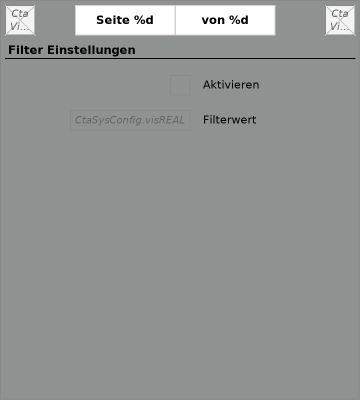
VISUALIZATION VIS_SENSOR_PARAMETER_FILTER  // 360x400
VAR_INPUT
  	ITF_SENSORIN	:	ITF_SENSOR;
END_VAR
VAR
    uiPage  :   UINT;
    uiMin   :   UINT    := 0;
    uiMax   :   UINT    := 0;
END_VAR
    Image (5,5 30x30), invisible if: uiPage = uiMin, image: CtaVisSymbols.ImagePool.arrow-left_square
        OnMouseClick: execute {
            uiPage := uiPage - 1;
            IF uiPage <= uiMin THEN
                uiPage := uiMin;
            END_IF;
        }
    Image (325,5 30x30), invisible if: uiPage = uiMax, image: CtaVisSymbols.ImagePool.arrow-right_square
        OnMouseClick: execute {
            uiPage := uiPage + 1;
            IF uiPage >= uiMax THEN
                uiPage := uiMax;
            END_IF;
        }
    Frame (0,40 360x360), frame switch variable: uiPage
        shows VIS_SENSOR_PARAMETER_FILTER_1(ITF_SENSORIN := ITF_SENSORIN)
        shows AT_ParameterIO1(ITF_Parameter := ITF_Parameter)
    Textfield (175,5 100x30), "von %d", text variable: uiMax
    Textfield (75,5 100x30), "Seite %d", text variable: uiPage
END_VISUALIZATION

// 40 Visualizations/POPUP/PARAMETER/SENSOR_Filter/VIS_SENSOR_PARAMETER_FILTER_1
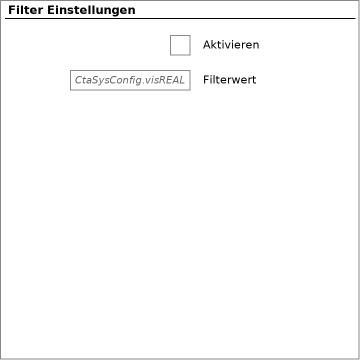
VISUALIZATION VIS_SENSOR_PARAMETER_FILTER_1  // 360x360
VAR_INPUT
   	ITF_SENSORIN	:	ITF_SENSOR;
END_VAR
    Label (5,0 350x20), "Filter Einstellungen"
    Line (5,18) (355,18)
    Frame (170,35 20x20)
        shows CtaSysConfig.visBOOL(visfbBOOLIn := ITF_SENSORIN.P_scFilter_fbxEnabled)
    Label (200,35 150x20), "Aktivieren"
    Frame (70,70 120x20)
        shows CtaSysConfig.visREAL(visfbREALIn := ITF_SENSORIN.P_scFilter_fbrValue)
    Label (200,70 150x20), "Filterwert"
END_VISUALIZATION

// 40 Visualizations/POPUP/PARAMETER/SENSOR_InfluxDb/VIS_SENSOR_PARAMETER_TRENDLOG
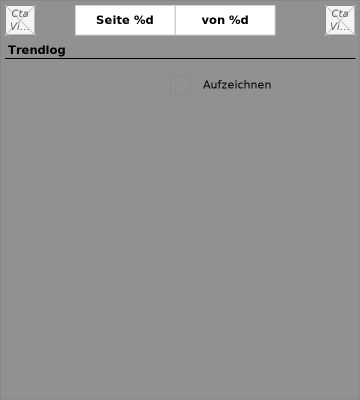
VISUALIZATION VIS_SENSOR_PARAMETER_TRENDLOG  // 360x400
VAR_INPUT
   	ITF_SENSORIN	:	ITF_SENSOR;
END_VAR
VAR
    uiPage  :   UINT;
    uiMin   :   UINT    := 0;
    uiMax   :   UINT    := 0;
END_VAR
    Image (5,5 30x30), invisible if: uiPage = uiMin, image: CtaVisSymbols.ImagePool.arrow-left_square
        OnMouseClick: execute {
            uiPage := uiPage - 1;
            IF uiPage <= uiMin THEN
                uiPage := uiMin;
            END_IF;
        }
    Image (325,5 30x30), invisible if: uiPage = uiMax, image: CtaVisSymbols.ImagePool.arrow-right_square
        OnMouseClick: execute {
            uiPage := uiPage + 1;
            IF uiPage >= uiMax THEN
                uiPage := uiMax;
            END_IF;
        }
    Frame (0,40 360x360), frame switch variable: uiPage
        shows VIS_SENSOR_PARAMETER_TRENDLOG0(ITF_SENSORIN := ITF_SENSORIN)
        shows AT_ParameterIO1(ITF_Parameter := ITF_Parameter)
        pReferences[0]: ITF_Parameter=ITF_Parameter
    Textfield (75,5 100x30), "Seite %d", text variable: uiPage
    Textfield (175,5 100x30), "von %d", text variable: uiMax
END_VISUALIZATION

// 40 Visualizations/POPUP/PARAMETER/SENSOR_InfluxDb/VIS_SENSOR_PARAMETER_TRENDLOG0
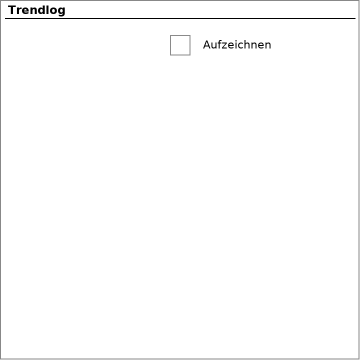
VISUALIZATION VIS_SENSOR_PARAMETER_TRENDLOG0  // 360x360
VAR_INPUT
    ITF_SENSORIN	:	ITF_SENSOR;
END_VAR
    Frame (170,35 20x20)
        shows CtaSysConfig.visBOOL(visfbBOOLIn := ITF_SENSORIN.P_scInfluxDb_fbxEnable)
    Label (200,35 150x20), "Aufzeichnen"
    Label (5,0 350x20), "Trendlog"
    Line (5,18) (355,18)
END_VISUALIZATION

// 40 Visualizations/POPUP/PARAMETER/SENSOR_ReportManagement/Sensor_LowWarning_Param
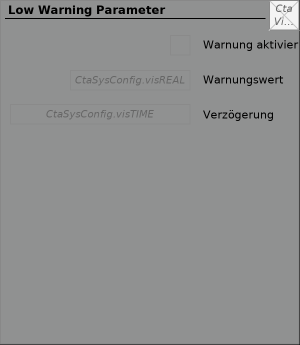
VISUALIZATION Sensor_LowWarning_Param  // 300x345
VAR_INPUT
	ITF_SENSORIN	:	ITF_SENSOR;
END_VAR
VAR_IN_OUT
    xShow   :   BOOL;
END_VAR
    Rectangle (0,0 300x345)
    Image (269,0 30x30), image: CtaVisSymbols.ImagePool.close_solo_black
        OnMouseClick: execute { xShow := FALSE; }
    Label (5,0 198x20), "Low Warning Parameter"
    Line (5,18) (265,18)
    Label (200,35 100x20), "Warnung aktiviert"
    Frame (170,35 20x20)
        shows CtaSysConfig.visBOOL(visfbBOOLIn := ITF_SENSORIN.P_scLoWarning_fbxDoesWarning)
    Label (200,70 100x20), "Warnungswert"
    Frame (70,70 120x20), invisible if: (ITF_SENSORIN.proValueInputType = enInputType.DigitalInput) OR (ITF_SENSORIN.proValueInputType = enInputType.Digital_ITF_Input)
        shows CtaSysConfig.visREAL(visfbREALIn := ITF_SENSORIN.P_scLoWarning_fbrValue)
    Label (200,105 100x20), "Verzögerung"
    Frame (10,104 180x20)
        shows CtaSysConfig.visTIME(visfbTIMEIn := ITF_SENSORIN.P_scLoWarning_fbtDelayTillWarning)
END_VISUALIZATION

// 40 Visualizations/ICON/SENSOR_FLAT/SENSOR_FLAT_TXT_RIGHT/ABOVE/VIS_SENSOR_FLAT_RigthAboveCheckQuerry
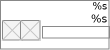
VISUALIZATION VIS_SENSOR_FLAT_RigthAboveCheckQuerry  // 110x50
VAR_INPUT
    ITF_SENSOR_IN   :   ITF_SENSOR;
	stExklParameter	:	STRING [40];
END_VAR
    Frame (0,0 110x50)
        shows VIS_SENSOR_FLAT_RigthAboveCheckIsEnabled(ITF_SENSOR_IN := ITF_SENSOR_IN, stExklParameter := stExklParameter)
END_VISUALIZATION

// 40 Visualizations/ICON/SENSOR_ROUND/SENSOR_ROUNF_TXT_LEFT/ABOVE/VIS_SENSOR_ROUND_LEFT_ABOVE
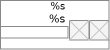
VISUALIZATION VIS_SENSOR_ROUND_LEFT_ABOVE  // 110x50
VAR_INPUT
    ITF_SENSOR_IN   :   ITF_SENSOR;	
END_VAR
VAR_INPUT CONSTANT	
	stExklParameter	:	STRING [40] := ' ';	
END_VAR
VAR CONSTANT
	uiIconnr		:	UINT := 6;
END_VAR
    Frame (0,0 110x50), invisible if: NOT fcCheckQuerryAndIconReturn(_ITF_IN := ITF_SENSOR_IN, _uiIconNr_IN := uiIconNr)
        shows VIS_SENSOR_ROUND_LeftAboveCheckQuerry(ITF_SENSOR_IN := ITF_SENSOR_IN, stExklParameter := stExklParameter)
END_VISUALIZATION

// 40 Visualizations/ICON/SENSOR_ROUND/SENSOR_ROUNF_TXT_LEFT/ABOVE/VIS_SENSOR_ROUND_LeftAboveCheckIsEnabled
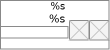
VISUALIZATION VIS_SENSOR_ROUND_LeftAboveCheckIsEnabled  // 110x50
VAR_INPUT
    ITF_SENSOR_IN   :   ITF_SENSOR;
	stExklParameter	:	STRING [40];	
END_VAR
    Frame (69,20 40x20), invisible if: NOT ITF_SENSOR_IN.proIsEnabled
        shows SensorRound(ITF_SENSORIN := ITF_SENSOR_IN)
    Frame (0,0 68x40), invisible if: NOT ITF_SENSOR_IN.proIsEnabled
        shows ValueUpDwn(ITF_SENSORIN := ITF_SENSOR_IN, uiTextAusrichtung := 6)
    Rectangle (0,0 110x50)
        OnMouseClick:  Dialog=POPUP_SENSOR, Parameters={stExklParameter: stExklParameter, ITF_SENSORIN: ITF_SENSOR_IN, uiPopUpGruppe: 0}, OpenCentered=True
END_VISUALIZATION

// 40 Visualizations/ICON/SENSOR_ROUND/SENSOR_ROUNF_TXT_LEFT/ABOVE/VIS_SENSOR_ROUND_LeftAboveCheckQuerry
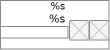
VISUALIZATION VIS_SENSOR_ROUND_LeftAboveCheckQuerry  // 110x50
VAR_INPUT
    ITF_SENSOR_IN   :   ITF_SENSOR;
	stExklParameter	:	STRING [40];	
END_VAR
    Frame (0,0 110x50)
        shows VIS_SENSOR_ROUND_LeftAboveCheckIsEnabled(ITF_SENSOR_IN := ITF_SENSOR_IN, stExklParameter := stExklParameter)
END_VISUALIZATION

// 40 Visualizations/ICON/SENSOR_ROUND/SENSOR_ROUND_TXT_RIGHT/ABOVE/VIS_SENSOR_ROUND_RIGHT_ABOVE
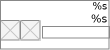
VISUALIZATION VIS_SENSOR_ROUND_RIGHT_ABOVE  // 110x50
VAR_INPUT
    ITF_SENSOR_IN   :   ITF_SENSOR;	
END_VAR
VAR_INPUT CONSTANT	
	stExklParameter	:	STRING [40] := ' ';	
END_VAR
VAR CONSTANT
	uiIconNr		:	UINT := 4;
END_VAR
    Frame (0,0 110x50), invisible if: NOT fcCheckQuerryAndIconReturn(_ITF_IN := ITF_SENSOR_IN, _uiIconNr_IN := uiIconNr)
        shows VIS_SENSOR_ROUND_RightAboveCheckQuerry(ITF_SENSOR_IN := ITF_SENSOR_IN, stExklParameter := stExklParameter)
END_VISUALIZATION

// 40 Visualizations/ICON/SENSOR_ROUND/SENSOR_ROUND_TXT_RIGHT/ABOVE/VIS_SENSOR_ROUND_RightAboveCheckIsEnabled
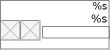
VISUALIZATION VIS_SENSOR_ROUND_RightAboveCheckIsEnabled  // 110x50
VAR_INPUT
    ITF_SENSOR_IN   :   ITF_SENSOR;
	stExklParameter	:	STRING [40];	
END_VAR
    Frame (0,20 40x20), invisible if: NOT ITF_SENSOR_IN.proIsEnabled
        shows SensorRound(ITF_SENSORIN := ITF_SENSOR_IN)
    Frame (42,0 68x40), invisible if: NOT ITF_SENSOR_IN.proIsEnabled
        shows ValueUpDwn(ITF_SENSORIN := ITF_SENSOR_IN, uiTextAusrichtung := 4)
    Rectangle (0,0 110x50)
        OnMouseClick:  Dialog=POPUP_SENSOR, Parameters={stExklParameter: stExklParameter, ITF_SENSORIN: ITF_SENSOR_IN, uiPopUpGruppe: 0}, OpenCentered=True
END_VISUALIZATION

// 40 Visualizations/ICON/SENSOR_ROUND/SENSOR_ROUND_TXT_RIGHT/ABOVE/VIS_SENSOR_ROUND_RightAboveCheckQuerry
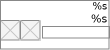
VISUALIZATION VIS_SENSOR_ROUND_RightAboveCheckQuerry  // 110x50
VAR_INPUT
    ITF_SENSOR_IN   :   ITF_SENSOR;
	stExklParameter	:	STRING [40];	
END_VAR
    Frame (0,0 110x50)
        shows VIS_SENSOR_ROUND_RightAboveCheckIsEnabled(ITF_SENSOR_IN := ITF_SENSOR_IN, stExklParameter := stExklParameter)
END_VISUALIZATION

// 40 Visualizations/ICON/SENSOR_FLAT/SENSOR_FLAT_TXT_RIGHT/BELOW/VIS_SENSOR_FLAT_RIGHT_BELOW
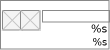
VISUALIZATION VIS_SENSOR_FLAT_RIGHT_BELOW  // 110x50
VAR_INPUT
    ITF_SENSOR_IN   :   ITF_SENSOR;	
END_VAR
VAR_INPUT CONSTANT	
	stExklParameter	:	STRING [40] := ' ';	
END_VAR
VAR CONSTANT
	uiIconNr		:	UINT := 3;
END_VAR
    Frame (0,0 110x50), invisible if: NOT fcCheckQuerryAndIconReturn(_ITF_IN := ITF_SENSOR_IN, _uiIconNr_IN := uiIconNr)
        shows VIS_SENSOR_FLAT_RigthBelowCheckQuerry(ITF_SENSOR_IN := ITF_SENSOR_IN, stExklParameter := stExklParameter)
END_VISUALIZATION

// 40 Visualizations/ICON/SENSOR_FLAT/SENSOR_FLAT_TXT_RIGHT/BELOW/VIS_SENSOR_FLAT_RigthBelowCheckIsEnabled
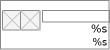
VISUALIZATION VIS_SENSOR_FLAT_RigthBelowCheckIsEnabled  // 110x50
VAR_INPUT
    ITF_SENSOR_IN   :   ITF_SENSOR;
	stExklParameter	:	STRING [40];	
END_VAR
    Frame (2,10 38x20), invisible if: NOT ITF_SENSOR_IN.proIsEnabled
        shows SensorFlat(ITF_SENSORIN := ITF_SENSOR_IN)
    Frame (42,10 68x40), invisible if: NOT ITF_SENSOR_IN.proIsEnabled
        shows ValueDwnUp(ITF_SENSORIN := ITF_SENSOR_IN, uiTextAusrichtung := 4)
    Rectangle (0,0 110x50)
        OnMouseClick:  Dialog=POPUP_SENSOR, Parameters={stExklParameter: stExklParameter, ITF_SENSORIN: ITF_SENSOR_IN, uiPopUpGruppe: 0}, OpenCentered=True
END_VISUALIZATION

// 40 Visualizations/ICON/SENSOR_FLAT/SENSOR_FLAT_TXT_RIGHT/BELOW/VIS_SENSOR_FLAT_RigthBelowCheckQuerry
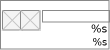
VISUALIZATION VIS_SENSOR_FLAT_RigthBelowCheckQuerry  // 110x50
VAR_INPUT
    ITF_SENSOR_IN   :   ITF_SENSOR;	
	stExklParameter	:	STRING [40];	
END_VAR
    Frame (0,0 110x50)
        shows VIS_SENSOR_FLAT_RigthBelowCheckIsEnabled(ITF_SENSOR_IN := ITF_SENSOR_IN, stExklParameter := stExklParameter)
END_VISUALIZATION

// 40 Visualizations/ICON/SENSOR_ROUND/SENSOR_ROUND_TXT_RIGHT/BELOW/VIS_SENSOR_ROUND_RIGHT_BELOW
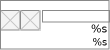
VISUALIZATION VIS_SENSOR_ROUND_RIGHT_BELOW  // 110x50
VAR_INPUT
    ITF_SENSOR_IN   :   ITF_SENSOR;	
END_VAR
VAR_INPUT CONSTANT	
	stExklParameter	:	STRING [40] := ' ';	
END_VAR
VAR CONSTANT
	uiIconNr		:	UINT := 5;
END_VAR
    Frame (0,0 110x50), invisible if: NOT fcCheckQuerryAndIconReturn(_ITF_IN := ITF_SENSOR_IN, _uiIconNr_IN := uiIconNr)
        shows VIS_SENSOR_ROUND_RightBelowCheckQuerry(ITF_SENSOR_IN := ITF_SENSOR_IN, stExklParameter := stExklParameter)
END_VISUALIZATION

// 40 Visualizations/ICON/SENSOR_BASE/ICON/Value/ValueDwnUp
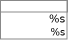
VISUALIZATION ValueDwnUp  // 68x40
VAR_INPUT
    ITF_SENSORIN   :   ITF_SENSOR;	
END_VAR
VAR_INPUT CONSTANT
    uiTextAusrichtung   : UINT := 4;    // 0 = Oben links | 1 = Horizontal zentriert | 2 = Rechts | 4 = Vertikal zentriert | 8 = Unten
END_VAR
    Frame (0,0 68x12)
        shows CtaSysSensorReCalculation.ValueRC(ITF_SENSOR_RE_CALCULATE := ITF_SENSORIN.ITF_RC, uiTextAusrichtung := uiTextAusrichtung)
    Textfield (0,13 68x12), "%s", text variable: ITF_SENSORIN.proSoftwareValue
        p3718999670: uiTextAusrichtung
    Textfield (0,26 68x12), "%s", text variable: ITF_SENSORIN.proGetBMK, invisible if: ITF_SENSORIN.proNoBmkInList
        p3718999670: uiTextAusrichtung
END_VISUALIZATION

// 40 Visualizations/ICON/SENSOR_BASE/ICON/Round/SensorRound
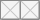
VISUALIZATION SensorRound  // 40x20
VAR_INPUT
    ITF_SENSORIN   :   ITF_SENSOR;	
END_VAR
    Ellipse (10,0 20x20), colour toggle: ITF_SENSORIN.proAcknowlege, invisible if: ITF_SENSORIN.proIsError
    Ellipse (10,0 20x20), colour toggle: ITF_SENSORIN.proIsError
    Image (0,0 20x20), invisible if: NOT ITF_SENSORIN.proIsWarning, image: CtaVisSymbols.ImagePool.CtaWarning
    Image (20,0 20x20), invisible if: NOT ITF_SENSORIN.proIsHandOnOrOff, image: CtaVisSymbols.ImagePool.front_hand_Yellow
    Image (20,0 20x20), invisible if: NOT ITF_SENSORIN.proHandOff, image: CtaVisSymbols.ImagePool.front_hand_Yellow_Off
END_VISUALIZATION

// 40 Visualizations/ICON/SENSOR_ROUND/SENSOR_ROUND_TXT_RIGHT/BELOW/VIS_SENSOR_ROUND_RightBelowCheckQuerry
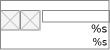
VISUALIZATION VIS_SENSOR_ROUND_RightBelowCheckQuerry  // 110x50
VAR_INPUT
    ITF_SENSOR_IN   :   ITF_SENSOR;
	stExklParameter	:	STRING [40];	
END_VAR
    Frame (0,0 110x50)
        shows VIS_SENSOR_ROUND_RightBelowCheckIsEnabled(ITF_SENSOR_IN := ITF_SENSOR_IN, stExklParameter := stExklParameter)
END_VISUALIZATION

// 40 Visualizations/ICON/SENSOR_ROUND/SENSOR_ROUND_TXT_RIGHT/BELOW/VIS_SENSOR_ROUND_RightBelowCheckIsEnabled
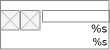
VISUALIZATION VIS_SENSOR_ROUND_RightBelowCheckIsEnabled  // 110x50
VAR_INPUT
    ITF_SENSOR_IN   :   ITF_SENSOR;
	stExklParameter	:	STRING [40];	
END_VAR
    Frame (0,10 40x20), invisible if: NOT ITF_SENSOR_IN.proIsEnabled
        shows SensorRound(ITF_SENSORIN := ITF_SENSOR_IN)
    Frame (42,10 68x40), invisible if: NOT ITF_SENSOR_IN.proIsEnabled
        shows ValueDwnUp(ITF_SENSORIN := ITF_SENSOR_IN, uiTextAusrichtung := 4)
    Rectangle (0,0 110x50)
        OnMouseClick:  Dialog=POPUP_SENSOR, Parameters={stExklParameter: , ITF_SENSORIN: ITF_SENSOR_IN, uiPopUpGruppe: 0}, OpenCentered=True
END_VISUALIZATION

// 40 Visualizations/ICON/SENSOR_ROUND/SENSOR_ROUNF_TXT_LEFT/BELOW/VIS_SENSOR_ROUND_LEFT_BELOW
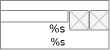
VISUALIZATION VIS_SENSOR_ROUND_LEFT_BELOW  // 110x50
VAR_INPUT
    ITF_SENSOR_IN   :   ITF_SENSOR;	
END_VAR
VAR_INPUT CONSTANT	
	stExklParameter	:	STRING [40] := ' ';	
END_VAR
VAR CONSTANT
	uiIconnr		:	UINT := 7;
END_VAR
    Frame (0,0 110x50), invisible if: NOT fcCheckQuerryAndIconReturn(_ITF_IN := ITF_SENSOR_IN, _uiIconNr_IN := uiIconNr)
        shows VIS_SENSOR_ROUND_LeftBelowCheckQuerry(ITF_SENSOR_IN := ITF_SENSOR_IN, stExklParameter := stExklParameter)
END_VISUALIZATION

// 40 Visualizations/ICON/SENSOR_ROUND/SENSOR_ROUNF_TXT_LEFT/BELOW/VIS_SENSOR_ROUND_LeftBelowCheckIsEnabled
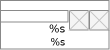
VISUALIZATION VIS_SENSOR_ROUND_LeftBelowCheckIsEnabled  // 110x50
VAR_INPUT
    ITF_SENSOR_IN   :   ITF_SENSOR;
	stExklParameter	:	STRING [40];	
END_VAR
    Frame (69,10 40x20), invisible if: NOT ITF_SENSOR_IN.proIsEnabled
        shows SensorRound(ITF_SENSORIN := ITF_SENSOR_IN)
    Frame (0,10 68x40), invisible if: NOT ITF_SENSOR_IN.proIsEnabled
        shows ValueDwnUp(ITF_SENSORIN := ITF_SENSOR_IN, uiTextAusrichtung := 6)
    Rectangle (0,0 110x50)
        OnMouseClick:  Dialog=POPUP_SENSOR, Parameters={stExklParameter: stExklParameter, ITF_SENSORIN: ITF_SENSOR_IN, uiPopUpGruppe: 0}, OpenCentered=True
END_VISUALIZATION

// 40 Visualizations/ICON/SENSOR_ROUND/SENSOR_ROUNF_TXT_LEFT/BELOW/VIS_SENSOR_ROUND_LeftBelowCheckQuerry
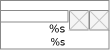
VISUALIZATION VIS_SENSOR_ROUND_LeftBelowCheckQuerry  // 110x50
VAR_INPUT
    ITF_SENSOR_IN   :   ITF_SENSOR;
	stExklParameter	:	STRING [40];	
END_VAR
    Frame (0,0 110x50)
        shows VIS_SENSOR_ROUND_LeftBelowCheckIsEnabled(ITF_SENSOR_IN := ITF_SENSOR_IN, stExklParameter := stExklParameter)
END_VISUALIZATION

// 40 Visualizations/POPUP/PARAMETER/IO_Parameter/VIS_SENSOR_IO_PARAMETER
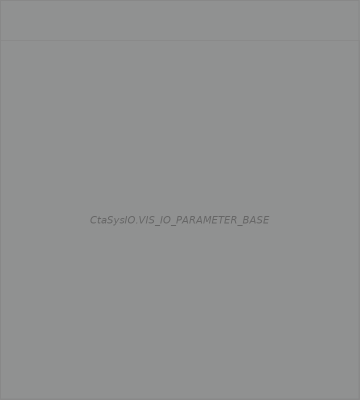
VISUALIZATION VIS_SENSOR_IO_PARAMETER  // 360x400
VAR_INPUT
    ITF_SENSORIN 	: 	ITF_SENSOR;
END_VAR
    Frame (0,40 360x360)
        shows CtaSysIO.VIS_IO_PARAMETER_BASE(ITF_IO_IN := ITF_SENSORIN.proSensorITF)
        shows AT_ParameterIO1(ITF_Parameter := ITF_Parameter)
END_VISUALIZATION

// 40 Visualizations/POPUP/OVERVIEW/VIS_SENSOR_OVERVIEW0
